// TIA Portal V20 export
// export: Created 2025-12-01T14:56:16.3794713Z, ExportSetting None, DisplayName Totally Integrated Automation Portal, DisplayVersion V20 Update 3, DisplayName TIA Portal Openness, DisplayVersion V20 Update 3, DisplayName TIA Portal Version Control Interface, DisplayVersion V20 Update 3, DisplayName STEP 7 Professional, DisplayVersion V20 Update 3, DisplayName STEP 7 Safety, DisplayVersion V20 Update 2, DisplayName WinCC Basic/Comfort/Advanced, DisplayVersion V20 Update 3, DisplayName WinCC Professional, DisplayVersion V20 Update 3, DisplayName WinCC Unified, DisplayVersion V20 Update 3
TYPE "ROUT_Reg_Etiqueta"
   STRUCT
      Anterior : UInt;   // posicion de la anterior etiqueta de la cola dentro del DB
      Posterior : UInt;   // posicion de la siguiente etiqueta de la cola dentro del DB
      CDB : ULInt;   // codigo de barras
      BIT_Orden : Array[0..50] of Bool;
   END_STRUCT;
END_TYPE
